// TIA Portal V19 export
DATA_BLOCK "UF DB"   // DB77
{ S7_Optimized_Access := 'FALSE' }
   VAR RETAIN
      "FORWARD FLUSH" : Int;
      "FILTRATION MODE" : Int;
      "AIR SCORING" : Int;
      "DRAIN BY GRAVITY" : Int;
      BACKWASH_1 : Int;
      BACKWASH_2 : Int;
      "FORWARD FLUSH_2" : Int;
      PV : Struct
         "FORWARD FLUSH" : Int;
         "FILTRATION MODE" : Int;
         "AIR SCORING" : Int;
         "DRAIN BY GRAVITY" : Int;
         BACKWASH_1 : Int;
         BACKWASH_2 : Int;
         "FORWARD FLUSH_2" : Int;
      END_STRUCT;
   END_VAR
BEGIN
END_DATA_BLOCK
